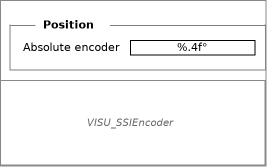
VISUALIZATION VISU_AxesElevationAxis_AbsoluteEncoder  // 267x167
VAR_IN_OUT
	ref : AxesElevationAxis;
    widget : AxesElevationAxisWidget;
END_VAR
    Frame (-5,80 270x85)
        shows VISU_SSIEncoder(ref := ref.parts.absoluteEncoder)
    Label (40,15 65x20), "Position"
    Polyline (110,25) (265,25) (265,70) (10,70) (10,25) (35,25)
    Label (20,40 105x15), "Absolute encoder"
    Rectangle (130,40 125x15), "%.4f°", text variable: ref.absoluteEncoderPosition.degrees.value
END_VISUALIZATION

(* stored: Version 1.1.0.1, ProductVersion 3.1.4019.2
   Visu VISU_AxesElevationAxis_AbsoluteEncoder: Id {deb4558d-2323-4679-9f4b-828a947b2db0} *)
